PROGRAM prgHP3
VAR
	fbWb2Com3						: FB_OCHSNER_Web2Com3;
	byHP1StateHeatProd		: BYTE;		//{#lynus.ag#()}
	lrHP1TWVtemp			: LREAL;	//{#lynus.ag#()}
	lrHP1TWRtemp			: LREAL;	//{#lynus.ag#()}
	lrHP1TQAtemp			: LREAL;	//{#lynus.ag#()}
	lrHP1TQEtemp			: LREAL;	//{#lynus.ag#()}
	lrHP1ThEnergykWh		: LREAL;	//{#lynus.ag#()}
	lrHP1ThEnergyMWh		: LREAL;	//{#lynus.ag#()}
	byHC1StateHC			: BYTE;		//{#lynus.ag#()}
	lrHC1OutTemp			: LREAL;	//{#lynus.ag#()}
	lrHC1OutTempAvg			: LREAL;	//{#lynus.ag#()}
	lrHC1RoomTemp			: LREAL;	//{#lynus.ag#()}
	lrHC1SPRoomTemp			: LREAL;	//{#lynus.ag#()}
	lrHC1PreFlowTemp		: LREAL;	//{#lynus.ag#()}
	lrHC1SPFlowTemp			: LREAL;	//{#lynus.ag#()}
END_VAR

fbWb2Com3(
	bStart:= TRUE, 
	tDelayRequest:= T#60S, 
	sHostname:= 'localhost', 
	bValidResult=> , 
	bBusy=> , 
	bError=> , 
	bDone=> , 
	hrErrorCode=> ,
	byHP1StateHeatProd => byHP1StateHeatProd,
	lrHP1TWVtemp => lrHP1TWVtemp,
	lrHP1TWRtemp => lrHP1TWRtemp,
	lrHP1TQAtemp => lrHP1TQAtemp,
	lrHP1TQEtemp => lrHP1TQEtemp,
	lrHP1ThEnergykWh => lrHP1ThEnergykWh,
	lrHP1ThEnergyMWh => lrHP1ThEnergyMWh,
	byHC1StateHC => byHC1StateHC,
	lrHC1OutTemp => lrHC1OutTemp,
	lrHC1OutTempAvg => lrHC1OutTempAvg,
	lrHC1RoomTemp => lrHC1RoomTemp,
	lrHC1SPRoomTemp => lrHC1SPRoomTemp,
	lrHC1PreFlowTemp => lrHC1PreFlowTemp,
	lrHC1SPFlowTemp => lrHC1SPFlowTemp);

END_PROGRAM

(* stored: Version 1.1.0.1, ProductVersion 3.1.4024.11
   POU prgHP3: Id {0f8df2b4-779b-48d6-8b9c-2293cb1fac8e}, SpecialFunc None *)
